FUNCTION_BLOCK Machine EXTENDS FB_Generic
VAR
END_VAR

SUPER^();

METHOD M_Aborting
VAR_INST
	bTest	: BOOL;
END_VAR
IF bTest THEN
	bTest := FALSE;
	M_StateComplete();
END_IF
END_METHOD

METHOD M_Execute
VAR_INST
	bTest	: BOOL;
END_VAR
IF bTest THEN
	bTest := FALSE;
	M_StateComplete();
END_IF
END_METHOD

METHOD M_StateComplete
SUPER^.M_StateComplete();
END_METHOD

END_FUNCTION_BLOCK

(* stored: Version 1.1.0.1
   POU Machine: Id {123c7c08-1b03-4b8d-8697-74435cc4f840}, SpecialFunc None
   Method M_Aborting: Id {9a7e0217-86ac-41de-9879-206cf8b6c989}
   Method M_Execute: Id {0418fa37-a42f-4b51-8426-e3bfff63d3fa}
   Method M_StateComplete: Id {dde11c87-adf4-44cf-ac55-3148d165f5a4} *)
